INTERFACE ITF_HighLevelSystem

PROPERTY eActivationStatus : ActivationStatus
GET
END_GET
SET
END_SET
END_PROPERTY

PROPERTY PUBLIC eCondition : HighLevelCondition
GET
END_GET
END_PROPERTY

PROPERTY PUBLIC nErrorID : UDINT
GET
END_GET
END_PROPERTY

END_INTERFACE

(* stored: Version 1.1.0.1, ProductVersion 3.1.4024.12
   Itf ITF_HighLevelSystem: Id {eca1f5f6-610b-45f5-b8b6-029235b687d2}
   Property eActivationStatus: Id {02c2974d-ea15-4b9b-b044-3477c47f2a68}
   Get Get: Id {deefed80-5355-44b5-a884-a08dd5eab10f}
   Set Set: Id {b9b41fd3-b9d0-4192-8102-2e6b553d5626}
   Property eCondition: Id {453906dd-cfca-4c2c-8fdd-7d983db9a8a0}
   Get Get: Id {ad14d373-2368-435d-81c1-88581710b5f2}
   Property nErrorID: Id {83326f54-283a-4ba6-a07d-7c14cde945ea}
   Get Get: Id {d92db387-7938-4179-8e21-f5e67a3bc76f} *)
